TYPE ST_HMI :
STRUCT
  nIrrLineSel  : UINT := 1;//at leat 1 robot line
END_STRUCT
END_TYPE

(* stored: Version 1.1.0.1, ProductVersion 3.1.4024.12
   DUT ST_HMI: Id {b27f09e8-ac45-4e71-adfb-086d626f648f} *)
